FUNCTION_BLOCK FB_FuseTest
VAR_INPUT
END_VAR
VAR_OUTPUT
END_VAR
VAR
	_chn1Basic : ITF_EL922x_ChannelBasic;
	_chn2Basic : ITF_EL922x_ChannelBasic;
	_chn1Extended : ITF_EL922x_ChannelExtended;
	_chn2Extended : ITF_EL922x_ChannelExtended;
END_VAR

METHOD GetDisabledBySwitch : BOOL
VAR_INPUT
END_VAR
IF _chn1Extended <> 0 THEN
	GetDisabledBySwitch := _chn1Extended.DisabledBySwitch;
END_IF
END_METHOD

METHOD METH : BOOL
VAR_INPUT
	chn1 : ITF_EL922x_ChannelBasic;
	chn2 : ITF_EL922x_ChannelBasic;
END_VAR
 VAR_INST
	 check : ITF_EL922x_ChannelBasic;
 END_VAR
_chn1Basic := chn1;
__QUERYINTERFACE(_chn1Basic, _chn1Extended);
_chn2Basic := chn2;
__QUERYINTERFACE(_chn2Basic, _chn2Extended);
END_METHOD

METHOD SwitchChannel1 : BOOL
VAR_INPUT
END_VAR
_chn1Basic.SwitchFuse();
END_METHOD

END_FUNCTION_BLOCK

(* stored: Version 1.1.0.1, ProductVersion 3.1.4024.5
   POU FB_FuseTest: Id {e47d6a39-c379-42ae-ae60-e27562337e6d}, SpecialFunc None
   Method GetDisabledBySwitch: Id {737118be-d9b4-4d0e-ab52-a5fa2e5cae34}
   Method METH: Id {f380b6b8-38a7-4257-b29b-b2e8fd5a4b74}
   Method SwitchChannel1: Id {93e7fa41-6392-4327-9a87-2b34e0dedc6a} *)
